// TIA Portal V16 export
// export: Created 2021-06-27T08:23:18.2377775Z, ExportSetting WithDefaults, DisplayName Totally Integrated Automation Portal, DisplayVersion V16 Update 4, DisplayName TIA Portal Version Control Interface, DisplayVersion V16 Update 2, DisplayName TIA Portal Openness, DisplayVersion V16 Update 4, DisplayName STEP 7 Professional, DisplayVersion V16 Update 4, DisplayName STEP 7 Safety, DisplayVersion V16, DisplayName WinCC Advanced, DisplayVersion V16 Update 4
FUNCTION "UpdateSensor" : Void   // FC7, F_FBD
{ S7_Optimized_Access := 'TRUE' }
VERSION : 0.1
// stored: AutoNumber true, IsIECCheckEnabled false, UDAEnableTagReadback false
   VAR_INPUT
      command : "SensorCommand";
   END_VAR
   VAR_OUTPUT
      ok : Bool;
   END_VAR
BEGIN

REGION Network 1
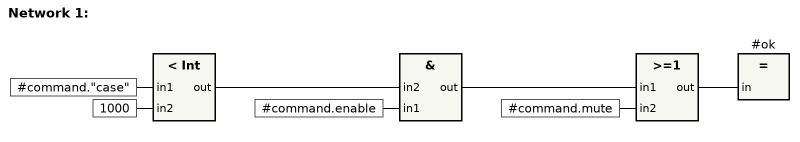
   #ok := ((#command."case" < 1000) AND #command.enable) OR #command.mute;
END_REGION
END_FUNCTION
